Omron CX-Programmer project NewProject (CX-Programmer 9.75)

# PLC NewPLC1: CP1L M

## Global symbols (name address type ; comment)
0.00 BOOL  ; BEL#1
0.01 BOOL  ; BEL#2
0.02 BOOL  ; BEL#3
100.00 BOOL  ; BUZZER#1
100.01 BOOL  ; BUZZER#2
100.02 BOOL  ; BUZZER#3
T0000 BOOL  ; RESET
W0.00 BOOL  ; PEMAIN#1
W0.01 BOOL  ; PEMAIN#2
W0.02 BOOL  ; PEMAIN#3

## Program NewProgram1 (cyclic task 0)

### Section Section1

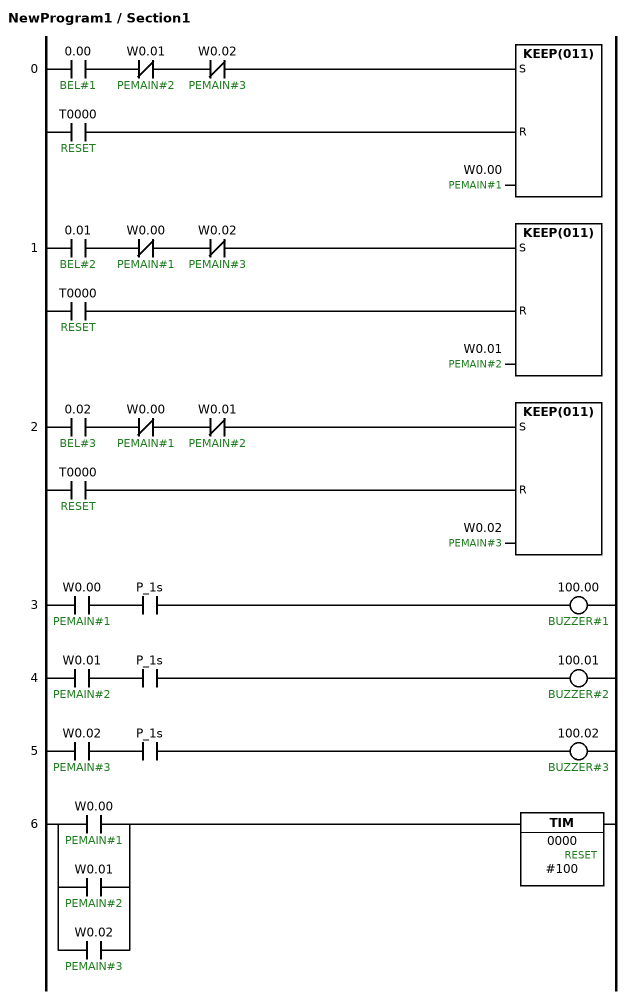
; rung 0
LD 0.00  ; BEL#1
ANDNOT W0.01  ; PEMAIN#2
ANDNOT W0.02  ; PEMAIN#3
LD T0000  ; RESET
KEEP(011) W0.00  ; PEMAIN#1
; rung 1
LD 0.01  ; BEL#2
ANDNOT W0.00  ; PEMAIN#1
ANDNOT W0.02  ; PEMAIN#3
LD T0000  ; RESET
KEEP(011) W0.01  ; PEMAIN#2
; rung 2
LD 0.02  ; BEL#3
ANDNOT W0.00  ; PEMAIN#1
ANDNOT W0.01  ; PEMAIN#2
LD T0000  ; RESET
KEEP(011) W0.02  ; PEMAIN#3
; rung 3
LD W0.00  ; PEMAIN#1
AND P_1s
OUT 100.00  ; BUZZER#1
; rung 4
LD W0.01  ; PEMAIN#2
AND P_1s
OUT 100.01  ; BUZZER#2
; rung 5
LD W0.02  ; PEMAIN#3
AND P_1s
OUT 100.02  ; BUZZER#3
; rung 6
LD W0.00  ; PEMAIN#1
OR W0.01  ; PEMAIN#2
OR W0.02  ; PEMAIN#3
TIM 0000 #100  ; RESET

### Section END
; rung 0
END(001)